// TwinCAT 3 PLC project CustomVisu_lib
// Title: CustomVisu_Frames
// Company: Chua Siang Poh
// Author: Chua Siang Poh
// ProjectVersion: 0.1.0
// ProgramVersion: 3.1.4020.10
// libraries:
//   Tc2_Standard, * (Beckhoff Automation GmbH)
//   Tc2_System, * (Beckhoff Automation GmbH)
//   Tc3_Module, * (Beckhoff Automation GmbH)
// project tree:
//   / GlobalTextList.TcGTLO, Visualization Manager.TcVMO (not stored)
//   Visualisation/TrendView/ M_TRENDVIEW_OBJECT.TcPOU
//   Visualisation/TrendView/VisuComponent/ TrendView.TcVIS, TrendView_PlotLineArea.TcVIS
// (motion and I/O tree: see PLC project motion_library)
// real-time tasks:
//   TASK PlcTask: cycle T#10ms, priority 20, ADS port 350

// ---- Visualisation/TrendView/M_TRENDVIEW_OBJECT.TcPOU
FUNCTION_BLOCK M_TRENDVIEW_OBJECT
VAR_INPUT
END_VAR
VAR_OUTPUT
END_VAR
VAR
	AXIS_Y_MAX : LREAL := 100;
	AXIS_Y_MIN : LREAL := -100;

	_CURRENT_DATA	: LREAL;
	_INTERNAL_DATA 	: ARRAY[0..BUFFER_WIDTH] OF LREAL;
	
	DISPLAY_Y_UNIT			: STRING(10);
	DISPLAY_TITLE			: STRING(30);
	DISPLAY_X_AXIS_LABEL	: STRING(25);
	DISPLAY_Y_AXIS_LABEL	: STRING(25);
	PLOT_WIDTH	: INT := 1;
	PLOT_POINTS : ARRAY[0..BUFFER_WIDTH] OF VisuElems.VisuStructPoint;
	
	_PLC_CYCLE_TICKS : UDINT := 10;
	_PLC_CYCLE_COUNT : UDINT;
END_VAR
VAR CONSTANT
	BUFFER_WIDTH : INT := 200;
	BUFFER_HEIGHT : INT := 200;
END_VAR

_PLC_CYCLE_COUNT := _PLC_CYCLE_COUNT + 1;
IF _PLC_CYCLE_COUNT >= _PLC_CYCLE_TICKS THEN
	_PLC_CYCLE_COUNT := 0;
	Tc2_System.MEMMOVE(ADR(_INTERNAL_DATA[1]), ADR(_INTERNAL_DATA[0]), BUFFER_WIDTH * 8);
	_INTERNAL_DATA[0] := _CURRENT_DATA;
	TRANSFORM_DATA();
END_IF

PROPERTY DISPLAY_UNIT : STRING(10)
GET
DISPLAY_UNIT := DISPLAY_Y_UNIT;
END_GET
SET
DISPLAY_Y_UNIT := DISPLAY_UNIT;
END_SET
END_PROPERTY

PROPERTY LINE_WIDTH : INT
GET
LINE_WIDTH := PLOT_WIDTH;
END_GET
SET
PLOT_WIDTH := LINE_WIDTH;
END_SET
END_PROPERTY

PROPERTY LOGGED_VALUE : LREAL
GET
LOGGED_VALUE := _CURRENT_DATA;
END_GET
SET
_CURRENT_DATA := LOGGED_VALUE;
END_SET
END_PROPERTY

PROPERTY TICKS : UDINT
GET
TICKS := _PLC_CYCLE_TICKS;
END_GET
SET
_PLC_CYCLE_TICKS := TICKS;
END_SET
END_PROPERTY

METHOD PROTECTED TRANSFORM_DATA
VAR_INPUT
END_VAR
VAR
	_I : INT;
END_VAR
FOR _I := 0 TO BUFFER_WIDTH BY 1 DO
	PLOT_POINTS[_I].iX := _I;
	PLOT_POINTS[_I].iY := LREAL_TO_INT(BUFFER_HEIGHT - ((_INTERNAL_DATA[_I] - AXIS_Y_MIN) / (AXIS_Y_MAX - AXIS_Y_MIN) * BUFFER_HEIGHT));
END_FOR
END_METHOD

PROPERTY X_AXIS_LABEL : STRING(25)
GET
X_AXIS_LABEL := DISPLAY_X_AXIS_LABEL;
END_GET
SET
DISPLAY_X_AXIS_LABEL := X_AXIS_LABEL;
END_SET
END_PROPERTY

PROPERTY Y_AXIS_LABEL : STRING(25)
GET
Y_AXIS_LABEL := DISPLAY_Y_AXIS_LABEL;
END_GET
SET
DISPLAY_Y_AXIS_LABEL := Y_AXIS_LABEL;
END_SET
END_PROPERTY

PROPERTY Y_MAX : LREAL
GET
Y_MAX := AXIS_Y_MAX;
END_GET
SET
AXIS_Y_MAX := Y_MAX;
END_SET
END_PROPERTY

PROPERTY Y_MIN : LREAL
GET
Y_MIN := AXIS_Y_MIN;
END_GET
SET
AXIS_Y_MIN := Y_MIN;
END_SET
END_PROPERTY

END_FUNCTION_BLOCK

// ---- GlobalTextList.TcGTLO
TEXTLIST GlobalTextList
  0 = '%.3f'
  1 = '%s'
END_TEXTLIST

// ---- Visualisation/TrendView/VisuComponent/TrendView.TcVIS
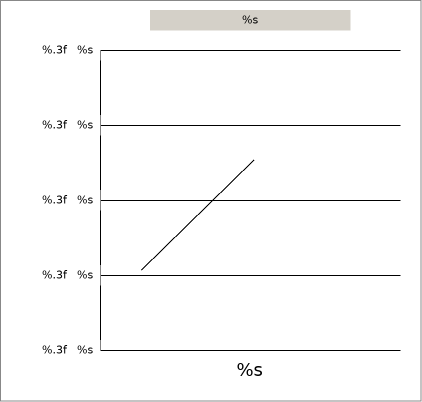
VISUALIZATION TrendView  // 422x402
VAR_IN_OUT
	PLC_IN : M_TRENDVIEW_OBJECT;
END_VAR
    Rectangle (0,0 420x400)
    Frame (100,50 300x300)
        shows TrendView_PlotLineArea(PLC_IN := PLC_IN)
    Line (100,50) (100,350)
    Line (100,350) (400,350)
    Line (100,200) (400,200)
    Line (100,125) (400,125)
    Line (100,275) (400,275)
    Line (100,50) (400,50)
    Textfield (20,40 50x20), "%.3f", text variable: PLC_IN.AXIS_Y_MAX, input disabled if: TRUE
    Textfield (70,40 30x20), "%s", text variable: PLC_IN.DISPLAY_Y_UNIT, input disabled if: TRUE
    Textfield (20,340 50x20), "%.3f", text variable: PLC_IN.AXIS_Y_MIN, input disabled if: TRUE
    Textfield (70,340 30x20), "%s", text variable: PLC_IN.DISPLAY_Y_UNIT, input disabled if: TRUE
    Textfield (200,360 100x20), "%s", text variable: PLC_IN.DISPLAY_X_AXIS_LABEL, input disabled if: TRUE
    Textfield (20,115 50x20), "%.3f", text variable: ((PLC_IN.AXIS_Y_MAX - PLC_IN.AXIS_Y_MIN) * 0.75) + PLC_IN.AXIS_Y_MIN, input disabled if: TRUE
    Textfield (70,115 30x20), "%s", text variable: PLC_IN.DISPLAY_Y_UNIT, input disabled if: TRUE
    Textfield (20,190 50x20), "%.3f", text variable: ((PLC_IN.AXIS_Y_MAX - PLC_IN.AXIS_Y_MIN) * 0.5) + PLC_IN.AXIS_Y_MIN, input disabled if: TRUE
    Textfield (70,190 30x20), "%s", text variable: PLC_IN.DISPLAY_Y_UNIT, input disabled if: TRUE
    Textfield (20,265 50x20), "%.3f", text variable: ((PLC_IN.AXIS_Y_MAX - PLC_IN.AXIS_Y_MIN) * 0.25) + PLC_IN.AXIS_Y_MIN, input disabled if: TRUE
    Textfield (70,265 30x20), "%s", text variable: PLC_IN.DISPLAY_Y_UNIT, input disabled if: TRUE
    Textfield (150,10 200x20), "%s", text variable: PLC_IN.DISPLAY_TITLE
END_VISUALIZATION

// ---- Visualisation/TrendView/VisuComponent/TrendView_PlotLineArea.TcVIS
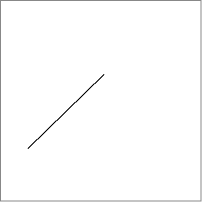
VISUALIZATION TrendView_PlotLineArea  // 202x202
VAR_IN_OUT
	PLC_IN : M_TRENDVIEW_OBJECT;
END_VAR
    Rectangle (0,0 200x200)
    Polyline (28,148) (104,74)
        p1271844420: PLC_IN.PLOT_WIDTH
        p3184209983: PLC_IN.BUFFER_WIDTH
        p1285906596: ADR(Plc_IN.PLOT_POINTS)
END_VISUALIZATION
